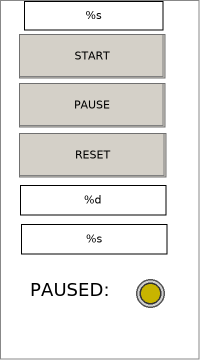
VISUALIZATION vSTATION_CONTROLLER  // 200x360
VAR_IN_OUT
	vSTATION : FB_STATION;
END_VAR
    Button (19,34 146x44), "START"
        OnMouseClick: execute { vSTATION.aSTART(); }
    Button (19,133 147x44), "RESET"
        OnMouseClick: execute { vSTATION.bRESET:=TRUE; }
    Rectangle (20,185 146x30), "%d", text variable: vSTATION.iSTATION_STATE
    Rectangle (21,224 146x30), "%s", text variable: vSTATION.sSTATION_STATE
    Button (19,83 146x44), "PAUSE"
        toggle vSTATION.bPAUSE
    Lamp1 (134,272 33x43), variable: vSTATION.bPAUSE, style: Lamp-Lamp1-Yellow
    Label (26,275 88x30), "PAUSED:"
    Rectangle (24,1 139x29), "%s", text variable: vSTATION.sName
END_VISUALIZATION

(* stored: Version 1.1.0.1, ProductVersion 3.1.4024.12
   Visu vSTATION_CONTROLLER: Id {27eb0ad1-51e5-4337-9208-f947727310d9} *)
